FUNCTION_BLOCK Demux8 (* Basic Function Block Type *)
  (* Standard: 61499-2 *)
  (* Version 0.0, 3/25/2015, jowelskop, nxtControl GmbH, Template *)
  PACKAGE Loytec.HVAC;
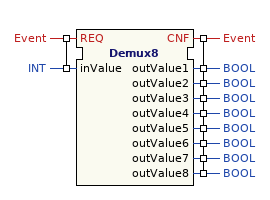
  EVENT_INPUT
    REQ WITH inValue; (* Normal Execution Request *)
  END_EVENT
  EVENT_OUTPUT
    CNF WITH outValue1, outValue2, outValue3, outValue4, outValue5, outValue6, outValue7, outValue8; (* Execution Confirmation *)
  END_EVENT
  VAR_INPUT
    inValue : INT; (* Input Value (from 1 to 8) *)
  END_VAR
  VAR_OUTPUT
    outValue1 : BOOL; (* Output TRUE if inValue = 1 *)
    outValue2 : BOOL; (* Output TRUE if inValue = 2 *)
    outValue3 : BOOL; (* Output TRUE if inValue = 3 *)
    outValue4 : BOOL; (* Output TRUE if inValue = 4 *)
    outValue5 : BOOL; (* Output TRUE if inValue = 5 *)
    outValue6 : BOOL; (* Output TRUE if inValue = 6 *)
    outValue7 : BOOL; (* Output TRUE if inValue = 7 *)
    outValue8 : BOOL; (* Output TRUE if inValue = 8 *)
  END_VAR
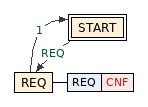
  EC_STATES
    START; (* Initial State *)
    REQ : REQ -> CNF; (* Normal execution *)
  END_STATES
  EC_TRANSITIONS
    START TO REQ := REQ;
    REQ TO START := 1;
  END_TRANSITIONS
  ALGORITHM REQ IN ST: (* Normally executed algorithm *)
IF inValue = 1 THEN outValue1 := TRUE;
	             ELSE outValue1 := FALSE;
END_IF ;

IF inValue = 2 THEN outValue2 := TRUE;
	             ELSE outValue2 := FALSE;
END_IF ;

IF inValue = 3 THEN outValue3 := TRUE;
	             ELSE outValue3 := FALSE;
END_IF ;

IF inValue = 4 THEN outValue4 := TRUE;
	             ELSE outValue4 := FALSE;
END_IF ;

IF inValue = 5 THEN outValue5 := TRUE;
	             ELSE outValue5 := FALSE;
END_IF ;

IF inValue = 6 THEN outValue6 := TRUE;
	             ELSE outValue6 := FALSE;
END_IF ;

IF inValue = 7 THEN outValue7 := TRUE;
	             ELSE outValue7 := FALSE;
END_IF ;

IF inValue = 8 THEN outValue8 := TRUE;
	             ELSE outValue8 := FALSE;
END_IF ;


;


;
  END_ALGORITHM
END_FUNCTION_BLOCK
